(* CoDeSys 2.3 export: E_TERMINAL.EXP *)

(* Data type *)
TYPE E_Terminal : (
	Beckhoff_KL3468 := 1, (* 0..10V *)
	Beckhoff_KL3208 := 2  (* PT1000, ...*)
);
END_TYPE
